(* IEC 61131-3 sources: CodesysTest/export/UN00 - Sharp Bagger/EM01 - Bagger Head/EM01_BaggerHead.pou/CurrentBagOpenRetryCount.prop, 2 files *)

(* ---- Get.pm.st ---- *)
(*#-#-#-#-#-#-#-#-#-#---Declaration---#-#-#-#-#-#-#-#-#-#-#-#-#*)

VAR
END_VAR
(*#-#-#-#-#-#-#-#-#-#---Implementation---#-#-#-#-#-#-#-#-#-#-#-#-#*)

CurrentBagOpenRetryCount := bagOpenRetryCount;

(* ---- Set.pm.st ---- *)
(*#-#-#-#-#-#-#-#-#-#---Declaration---#-#-#-#-#-#-#-#-#-#-#-#-#*)

VAR
END_VAR
(*#-#-#-#-#-#-#-#-#-#---Implementation---#-#-#-#-#-#-#-#-#-#-#-#-#*)

bagOpenRetryCount := CurrentBagOpenRetryCount;
